TYPE "SF_SafeBool"
VERSION : 0.1
   STRUCT
      Value { ExternalAccessible := 'False'; ExternalVisible := 'False'; ExternalWritable := 'False'} : Bool;
   END_STRUCT;

END_TYPE

